FUNCTION_BLOCK FB_VisuMessage IMPLEMENTS I_VisuMessage;


VAR	
	bInfo				: BOOL;
	bAlarm				: BOOL;
	bError				: BOOL;

	nMessageColor		: DWORD;
	_sMessageText_L1	: STRING;
	_sMessageText_L2	: STRING;

	stVisuOut			: ST_VisuMessage;


	sInfoMessage		: STRING;
	sInfoSequence		: STRING;
	nInfoState			: DINT;
	
	sCurrentSequence	: STRING;
	
	_sErrorMessage	: STRING;
	_sErrorSequence	: STRING;
	_nErrorState	: DINT;
	_nErrorCode		: DWORD;

	nColor_Green	: DWORD := 16#FF189E00;
	nColor_Yellow	: DWORD := 16#FFE6A000;
	nColor_Red		: DWORD := 16#FFFF0000;
	nColor_Black	: DWORD := 16#FF000000;


	_bAcknowledge	: BOOL;
	
	
	
END_VAR

METHOD CheckAknowledge : BOOL
VAR_INPUT
END_VAR



	CheckAknowledge := _bAcknowledge;
	  _bAcknowledge := FALSE;
END_METHOD

METHOD ClearAlarmMessage : BOOL
VAR_INPUT
END_VAR
END_METHOD

METHOD ClearAllMessages : BOOL
VAR_INPUT
END_VAR

	bError := FALSE;
	bInfo  := FALSE;
	
	ClearAllMessages := TRUE;
END_METHOD

METHOD ClearInfoMessage : BOOL
VAR_INPUT
END_VAR



	bInfo  := FALSE;
	
	ClearInfoMessage := TRUE;
END_METHOD

METHOD Cycle : BOOL
VAR_INPUT
	bAcknowledge	: BOOL;
END_VAR


	IF bAcknowledge THEN
		_bAcknowledge := TRUE;
	END_IF


	stVisuOut.bVisible_Box1_A := FALSE;
	stVisuOut.bVisible_Box1_B := FALSE;		


	IF bInfo THEN
		_sMessageText_L1 := CONCAT(sInfoMessage, ' - ');
		_sMessageText_L1 := CONCAT(_sMessageText_L1, sInfoSequence);
		
		IF nInfoState <> 0 THEN	
			_sMessageText_L1 := CONCAT(_sMessageText_L1, ' - State:');
			_sMessageText_L1 := CONCAT(_sMessageText_L1, DINT_TO_STRING(nInfoState));
		END_IF
		
		stVisuOut.bVisible_Box1_A := TRUE;
		stVisuOut.bVisible_Box1_B := FALSE;		
		
		stVisuOut.sMessage_L1_Box1.sText  := _sMessageText_L1;
		stVisuOut.sMessage_L1_Box1.nColor := nColor_Green;
	END_IF
	
	
	
//	IF bAlarm THEN
//		stVisuOut.sMessage_L1_Box1 := _sMessageText_L1;
//		stVisuOut.nColor_Box1   := nColor_Yellow;
//	END_IF

	
	
	
	IF bError THEN
		
		_sMessageText_L1 := CONCAT('Sequence: ' , _sErrorSequence);
		_sMessageText_L1 := CONCAT(_sMessageText_L1, ' - State:');
		_sMessageText_L1 := CONCAT(_sMessageText_L1, DINT_TO_STRING(_nErrorState));	
		

		_sMessageText_L2 := CONCAT('Error Message: ', _sErrorMessage);
		
		IF _nErrorCode > 0 THEN 
			_sMessageText_L2 := CONCAT(_sMessageText_L2,  ' - Error Code: ');
			_sMessageText_L2 := CONCAT(_sMessageText_L2, DWORD_TO_STRING(_nErrorCode));
		END_IF
	
	
		stVisuOut.bVisible_Box1_A := FALSE;
		stVisuOut.bVisible_Box1_B := TRUE;

		
		stVisuOut.sMessage_L1_Box1.sText  := _sMessageText_L1;
		stVisuOut.sMessage_L1_Box1.nColor := nColor_Red;
		
		stVisuOut.sMessage_L2_Box1.sText  := _sMessageText_L2;
		stVisuOut.sMessage_L2_Box1.nColor := nColor_Red;
		
	END_IF
END_METHOD

PROPERTY P_VisuOut : ST_VisuMessage
GET
P_VisuOut := stVisuOut;
END_GET
END_PROPERTY

METHOD SetAlarmMessage : BOOL
VAR_INPUT
	sMessage	: STRING;
END_VAR



	bError := FALSE;

	SetAlarmMessage := TRUE;
END_METHOD

METHOD SetErrorMessage : BOOL
VAR_INPUT
	sMessage	: STRING;
	sSequence	: STRING;
	nState		: DINT;
	nErrorCode	: DWORD;
END_VAR

	bError := TRUE;
	bInfo  := FALSE;

	_sErrorMessage	:= sMessage;
	_sErrorSequence	:= sSequence;
	
	sCurrentSequence := sSequence;
	
	_nErrorState	:= nState;
	_nErrorCode		:= nErrorCode;
	
	
	SetErrorMessage := TRUE;
END_METHOD

METHOD SetInfoMessage : BOOL
VAR_INPUT
	sMessage	: STRING;
	sSequence	: STRING;
	nState		: DINT;
END_VAR

	bInfo  := TRUE;
	bError := FALSE;

	
	sInfoMessage	 := sMessage;
	sInfoSequence	 := sSequence;
	sCurrentSequence := sSequence;
	nInfoState		 := nState;
	
	
	SetInfoMessage  := TRUE;
END_METHOD

METHOD StateUpdate : BOOL
VAR_INPUT
	nState		: DINT;
	sSequence	: STRING;
END_VAR



	IF sSequence = sCurrentSequence THEN

		nInfoState := nState;
		
	END_IF



	
	StateUpdate := TRUE;
END_METHOD

END_FUNCTION_BLOCK

(* stored: Version 1.1.0.1, ProductVersion 3.1.4024.13
   POU FB_VisuMessage: Id {e92c48ba-f99c-45ed-b9b0-3a62aa71a2d3}, SpecialFunc None
   Method CheckAknowledge: Id {9436697c-7f35-4fef-9b33-830a58cec987}
   Method ClearAlarmMessage: Id {c0e9be41-23e9-41b9-82a8-196bc003a1b7}
   Method ClearAllMessages: Id {35e25f7d-8b0c-4023-abac-66acd718138f}
   Method ClearInfoMessage: Id {df097ac0-df2c-4f68-ae90-410beb03a0ef}
   Method Cycle: Id {fcc8cddb-b11f-49ab-b551-f078f42bd903}
   Property P_VisuOut: Id {1974a4ef-c125-46ef-82d7-98e82bb579f3}
   Get Get: Id {457208bb-f21d-4043-92d8-c864e53d1cda}
   Method SetAlarmMessage: Id {c43c29ad-9b2d-446b-9ff8-79a5912a8888}
   Method SetErrorMessage: Id {87153b68-c59f-47bf-a767-6de0516f7002}
   Method SetInfoMessage: Id {960ca104-6f70-41e5-9a95-c4d290a917e9}
   Method StateUpdate: Id {5eca5a1f-6a9d-4b8b-a6fd-f32c7bf32d5e} *)
